TYPE "Bound_ShW"
VERSION : 0.1
   STRUCT
      Trigger : Bool;
      MainID : String[48];
      CarrierID : Int;
      Completed : Bool;
      Result : Int;
   END_STRUCT;

END_TYPE

